// Reverse sign of negative measurements (surplus) and output values >= 0
FUNCTION F_NormalizeSurplus : REAL
VAR_INPUT
    fIn: REAL;
END_VAR

IF fIn > 0 THEN
    // Cap any energy draw to 0
    F_NormalizeSurplus := 0;
ELSE
    // Reverse surplus to positive value
    F_NormalizeSurplus := fIn * -1;
END_IF

END_FUNCTION

(* stored: Version 1.1.0.1
   POU F_NormalizeSurplus: Id {3820aa7f-200f-463a-a983-f5607d4ae1d4}, SpecialFunc None *)
